{attribute 'hide'}
{attribute 'reflection'}
FUNCTION_BLOCK TInteger
VAR
    Value : INT;
END_VAR

{attribute 'TcRpcEnable'}
METHOD Inc : INT
VAR_INPUT
END_VAR
Value := Value + 1;
Inc := Value;
END_METHOD

METHOD Init
VAR_INPUT
    Value : INT;
END_VAR
THIS^.Value := Value;
END_METHOD

END_FUNCTION_BLOCK

(* stored: Version 1.1.0.1, ProductVersion 3.1.4024.4
   POU TInteger: Id {3c8577d3-012a-0947-1c69-6d02b1da422e}, SpecialFunc None
   Method Inc: Id {254ff61b-3caf-0007-3cf9-d6376a014065}
   Method Init: Id {3b590d3e-78a9-0a06-0a29-3c562a199e08} *)
